FUNCTION Next 
VAR_INPUT
END_VAR
VAR
END_VAR

//passe à l'étape suivante des cases dans le _4_Action_active
G_Match.iEtapeAction := G_Match.iEtapeAction + 1;

END_FUNCTION

(* stored: Version 1.1.0.1, ProductVersion 3.1.4024.12
   POU Next: Id {d3b22c90-bd98-4859-b303-dabbf9611a0d}, SpecialFunc None *)
